TYPE E_Mfr_LogLevel :
(
	eDebug		:= 0,
	eInfo		:= 1,
	eWarning	:= 2,
	eError		:= 3,
	eCritical	:= 4
);
END_TYPE

(* stored: Version 1.1.0.1
   DUT E_Mfr_LogLevel: Id {3f7a3d4d-85d3-41e3-8f7f-25d00ac1a9f3} *)
